TYPE ST_SelectStruct :
STRUCT
	id: DINT;
	username: STRING(199);
	password: STRING(199);
END_STRUCT
END_TYPE

(* stored: Version 1.1.0.1, ProductVersion 3.1.4024.4
   DUT ST_SelectStruct: Id {00f1fc49-a066-4ffd-afdd-4386dc99361b} *)
